// SIMATIC S7-200 project (STEP 7-Micro/WIN), CPU 224 REL 02.01

ORGANIZATION_BLOCK MAIN:OB1
TITLE=PROGRAM COMMENTS
BEGIN
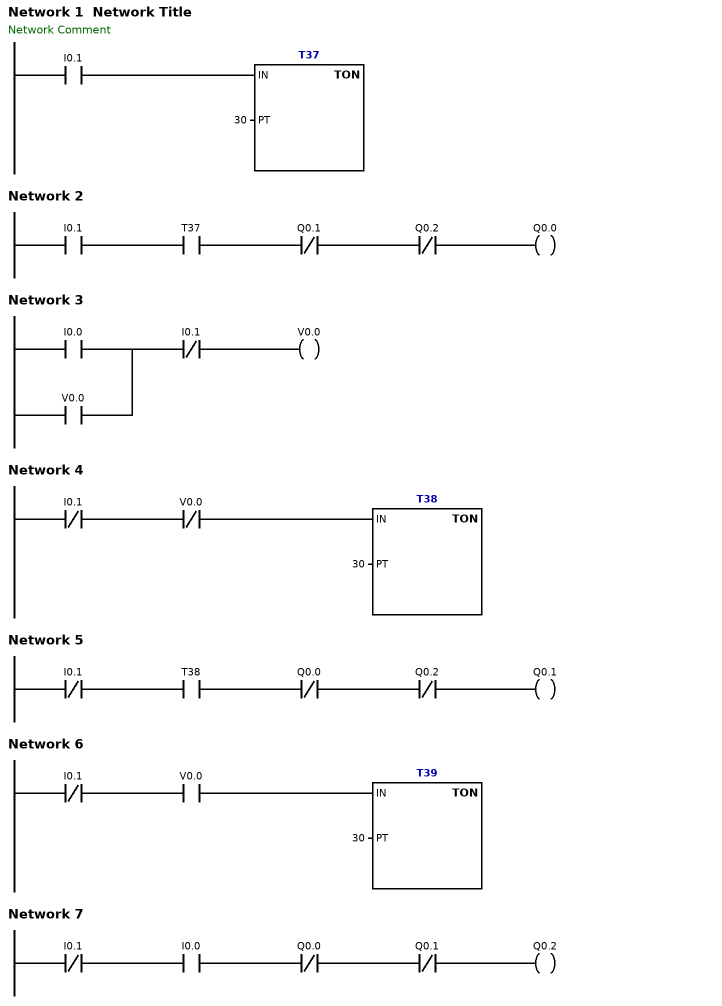
Network 1 // Network Title
// Network Comment
LD     I0.1
TON    T37, 30
Network 2
LD     I0.1
A      T37
AN     Q0.1
AN     Q0.2
=      Q0.0
Network 3
LD     I0.0
O      V0.0
AN     I0.1
=      V0.0
Network 4
LDN    I0.1
AN     V0.0
TON    T38, 30
Network 5
LDN    I0.1
A      T38
AN     Q0.0
AN     Q0.2
=      Q0.1
Network 6
LDN    I0.1
A      V0.0
TON    T39, 30
Network 7
LDN    I0.1
A      I0.0
AN     Q0.0
AN     Q0.1
=      Q0.2
END_ORGANIZATION_BLOCK
